FUNCTION_BLOCK FB_Flasher
VAR
	timON: TON;
	timOFF: TON;

END_VAR

VAR_INPUT
	timeVal:TIME;
	
END_VAR

VAR_OUTPUT
	q:BOOL;

END_VAR

//time on flasher
timON(	IN:= NOT timOFF.Q,
		PT:= timeVal
		);
		
q:= timON.Q;


//time off
timOFF(	IN:= timON.Q,
		PT:= timeVal
		);

END_FUNCTION_BLOCK

(* stored: Version 1.1.0.1, ProductVersion 3.1.4024.12
   POU FB_Flasher: Id {91d2bfd0-504b-4e5a-9e47-8efd9a85c590}, SpecialFunc None *)
